INTERFACE ITF_2_AMR EXTENDS ITF_1_Robot

PROPERTY ActualJointPosition : stJoint2
GET
END_GET
END_PROPERTY

PROPERTY ActualJointVelocity : stJoint2
GET
END_GET
END_PROPERTY

PROPERTY ActualTcpPose : stPose2D
GET
END_GET
END_PROPERTY

PROPERTY ActualTcpVelocity : stPose2D
GET
END_GET
END_PROPERTY

METHOD Dock : BOOL
VAR_INPUT
END_VAR
END_METHOD

PROPERTY IsDocked : BOOL
GET
END_GET
END_PROPERTY

METHOD NavigateToGoal : BOOL
  VAR_INPUT
    goal : STRING;
  END_VAR
END_METHOD

METHOD NavigateToPoint : BOOL
  VAR_INPUT
    point : stPose2D;
  END_VAR
END_METHOD

{warning 'Add property implementation'}
PROPERTY TargetReached : BOOL
GET
END_GET
SET
END_SET
END_PROPERTY

METHOD Undock : BOOL
  VAR_INPUT
  END_VAR
END_METHOD

END_INTERFACE

(* stored: Version 1.1.0.1, ProductVersion 3.1.4026.18
   Itf ITF_2_AMR: Id {46d1d572-82fe-4b3c-a5b8-9dc62cbaa12e}
   Property ActualJointPosition: Id {2deb01a8-8603-4d6d-b3b6-5ead78a8c2da}
   Get Get: Id {0cb3773a-7d8b-456f-a7e6-88106e5b8f49}
   Property ActualJointVelocity: Id {cf074f79-aa50-4fda-83f4-3c54291afca0}
   Get Get: Id {a33539de-f56c-471f-9ace-e2e7de977622}
   Property ActualTcpPose: Id {831ceed7-2617-41c1-8c18-8a215c121b7b}
   Get Get: Id {93f8d1ef-7924-4a2c-a53c-3c6b67f7af41}
   Property ActualTcpVelocity: Id {978d98cf-314d-4a06-bce6-c7862b54f7da}
   Get Get: Id {118a71d0-5d0a-4d44-82d2-e1740559cd71}
   Method Dock: Id {8a31a064-5d17-4519-bdc0-d55a86b86aa5}
   Property IsDocked: Id {b9186b89-8c8b-46b6-bd1b-dc333afe5375}
   Get Get: Id {61d4cdf3-33b8-4275-891c-244548dc4960}
   Method NavigateToGoal: Id {c2a8df64-60ad-4b7a-9b3f-5b0b6cd5e031}
   Method NavigateToPoint: Id {48f91d39-0773-4800-994b-b41b1d05a064}
   Property TargetReached: Id {884d6d0c-87d7-4a0b-bb70-b2a00f948294}
   Get Get: Id {4a3dd3c9-4383-4a54-8e9d-2410c9da3079}
   Set Set: Id {977c5a07-1875-42e2-b0a3-3e7cb7be0986}
   Method Undock: Id {b7f04aa5-1c68-4dc8-b065-6c8dd279892e} *)
